% RSLogix 500 project SERVO VALVE CONTROL_BAK046.RSS, saved by version 8.30.00.16 %
PROJECT "UNTITLED"    % processor: Bul.1763 MicroLogix 1100 Series B %

PROGRAM FILES
  LAD 2 "MAIN"  4 rungs
  LAD 3 "DIGITAL IO"  8 rungs
  LAD 4 "CONTROLS"  8 rungs
  LAD 5 "POSITION"  6 rungs

DATA FILES
  O0 OUTPUT  4 elements
  I1 INPUT  6 elements
  S2 STATUS  66 elements
  B3 BINARY  12 elements
  T4 TIMER  3 elements
  C5 COUNTER  1 elements
  R6 CONTROL  1 elements
  N7 INTEGER  2 elements
  F8 FLOAT  1 elements

LADDER 2 "MAIN"
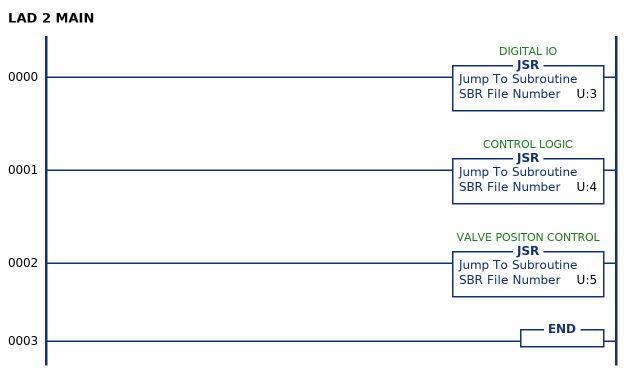
% Rung: 0 %
SOR JSR U:3 EOR
%   U:3  "DIGITAL IO" %
% Rung: 1 %
SOR JSR U:4 EOR
%   U:4  "CONTROL LOGIC" %
% Rung: 2 %
SOR JSR U:5 EOR
%   U:5  "VALVE POSITON CONTROL" %
% Rung: 3 %
SOR END EOR

LADDER 3 "DIGITAL IO"
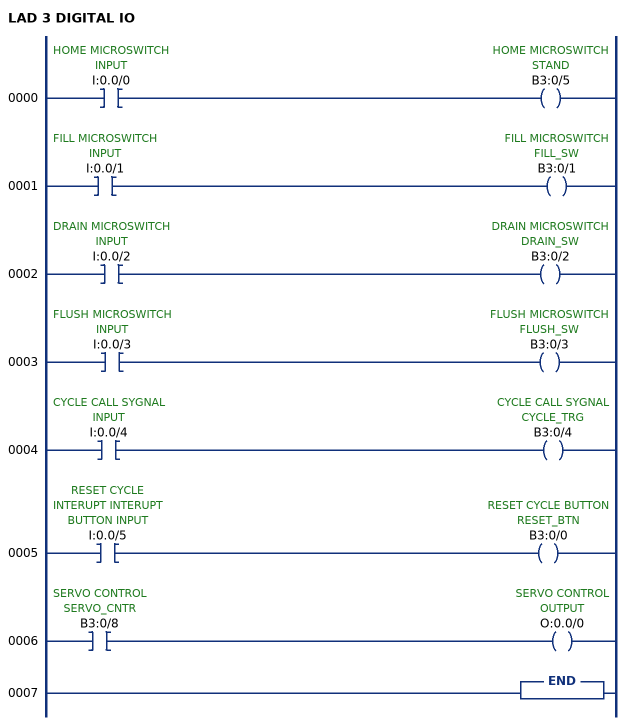
% Rung: 0 %
SOR XIC I:0.0/0 OTE B3:0/5 EOR
%   I:0.0/0  "HOME MICROSWITCH INPUT" %
%   B3:0/5  STAND  "HOME MICROSWITCH" %
% Rung: 1 %
SOR XIC I:0.0/1 OTE B3:0/1 EOR
%   I:0.0/1  "FILL MICROSWITCH INPUT" %
%   B3:0/1  FILL_SW  "FILL MICROSWITCH" %
% Rung: 2 %
SOR XIC I:0.0/2 OTE B3:0/2 EOR
%   I:0.0/2  "DRAIN MICROSWITCH INPUT" %
%   B3:0/2  DRAIN_SW  "DRAIN MICROSWITCH" %
% Rung: 3 %
SOR XIC I:0.0/3 OTE B3:0/3 EOR
%   I:0.0/3  "FLUSH MICROSWITCH INPUT" %
%   B3:0/3  FLUSH_SW  "FLUSH MICROSWITCH" %
% Rung: 4 %
SOR XIC I:0.0/4 OTE B3:0/4 EOR
%   I:0.0/4  "CYCLE CALL SYGNAL INPUT" %
%   B3:0/4  CYCLE_TRG  "CYCLE CALL SYGNAL" %
% Rung: 5 %
SOR XIC I:0.0/5 OTE B3:0/0 EOR
%   I:0.0/5  "RESET CYCLE INTERUPT INTERUPT BUTTON INPUT" %
%   B3:0/0  RESET_BTN  "RESET CYCLE BUTTON" %
% Rung: 6 %
SOR XIC B3:0/8 OTE O:0.0/0 EOR
%   B3:0/8  SERVO_CNTR  "SERVO CONTROL" %
%   O:0.0/0  "SERVO CONTROL OUTPUT" %
% Rung: 7 %
SOR END EOR

LADDER 4 "CONTROLS"
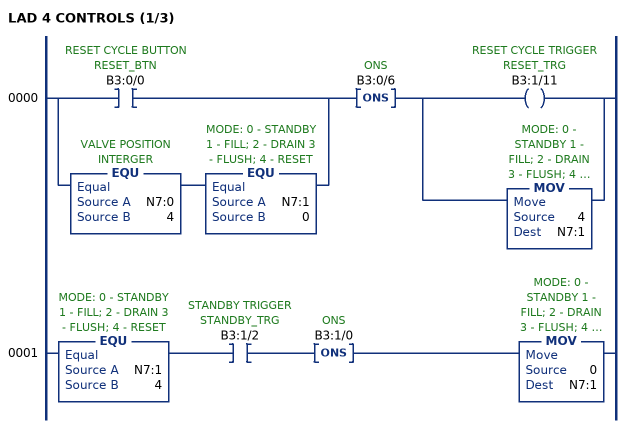
% Rung: 0 %
SOR BST XIC B3:0/0 NXB EQU N7:0 4 EQU N7:1 0 BND ONS B3:0/6 BST OTE B3:1/11 NXB MOV 4 N7:1 BND EOR
%   B3:0/0  RESET_BTN  "RESET CYCLE BUTTON" %
%   N7:0  "VALVE POSITION INTERGER" %
%   N7:1  "MODE: 0 - STANDBY 1 - FILL; 2 - DRAIN 3 - FLUSH; 4 - RESET" %
%   B3:0/6  "ONS" %
%   B3:1/11  RESET_TRG  "RESET CYCLE TRIGGER" %
% Rung: 1 %
SOR EQU N7:1 4 XIC B3:1/2 ONS B3:1/0 MOV 0 N7:1 EOR
%   N7:1  "MODE: 0 - STANDBY 1 - FILL; 2 - DRAIN 3 - FLUSH; 4 - RESET" %
%   B3:1/2  STANDBY_TRG  "STANDBY TRIGGER" %
%   B3:1/0  "ONS" %

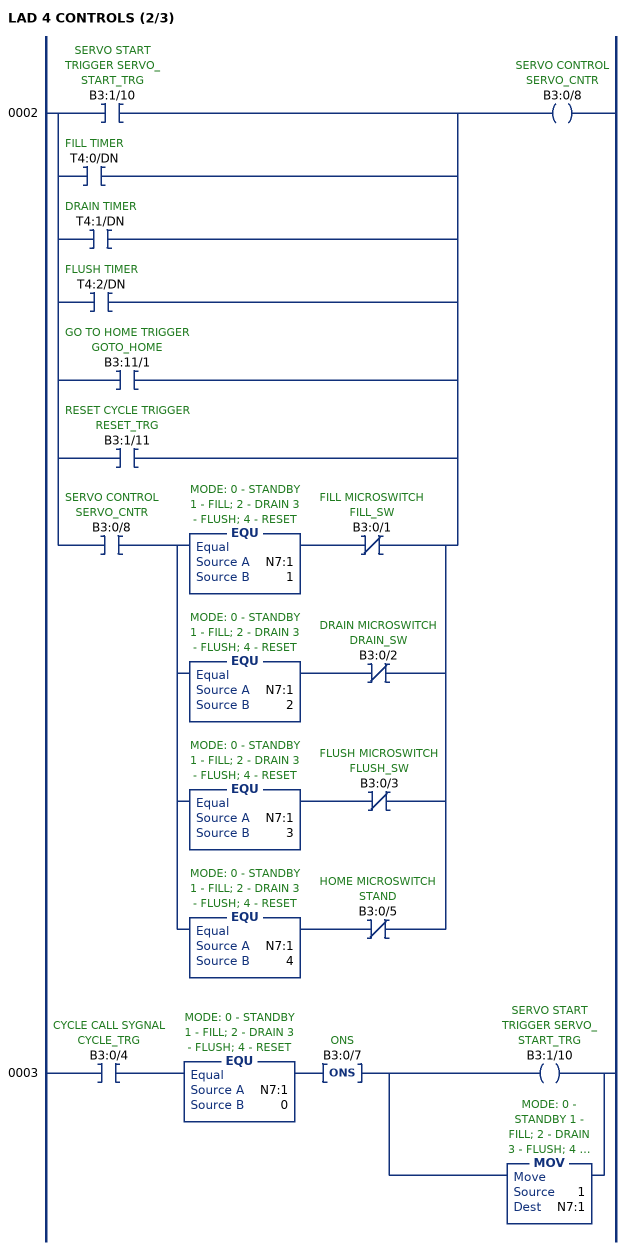
% Rung: 2 %
SOR BST BST XIC B3:1/10 NXB XIC T4:0/DN NXB XIC T4:1/DN NXB XIC T4:2/DN NXB XIC B3:11/1 NXB XIC B3:1/11 BND NXB XIC B3:0/8 BST EQU N7:1 1 XIO B3:0/1 NXB EQU N7:1 2 XIO B3:0/2 NXB EQU N7:1 3 XIO B3:0/3 NXB EQU N7:1 4 XIO B3:0/5 BND BND OTE B3:0/8 EOR
%   B3:1/10  SERVO_START_TRG  "SERVO START TRIGGER" %
%   T4:0  "FILL TIMER" %
%   T4:1  "DRAIN TIMER" %
%   T4:2  "FLUSH TIMER" %
%   B3:11/1  GOTO_HOME  "GO TO HOME TRIGGER" %
%   B3:1/11  RESET_TRG  "RESET CYCLE TRIGGER" %
%   B3:0/8  SERVO_CNTR  "SERVO CONTROL" %
%   N7:1  "MODE: 0 - STANDBY 1 - FILL; 2 - DRAIN 3 - FLUSH; 4 - RESET" %
%   B3:0/1  FILL_SW  "FILL MICROSWITCH" %
%   B3:0/2  DRAIN_SW  "DRAIN MICROSWITCH" %
%   B3:0/3  FLUSH_SW  "FLUSH MICROSWITCH" %
%   B3:0/5  STAND  "HOME MICROSWITCH" %
% Rung: 3 %
SOR XIC B3:0/4 EQU N7:1 0 ONS B3:0/7 BST OTE B3:1/10 NXB MOV 1 N7:1 BND EOR
%   B3:0/4  CYCLE_TRG  "CYCLE CALL SYGNAL" %
%   N7:1  "MODE: 0 - STANDBY 1 - FILL; 2 - DRAIN 3 - FLUSH; 4 - RESET" %
%   B3:0/7  "ONS" %
%   B3:1/10  SERVO_START_TRG  "SERVO START TRIGGER" %

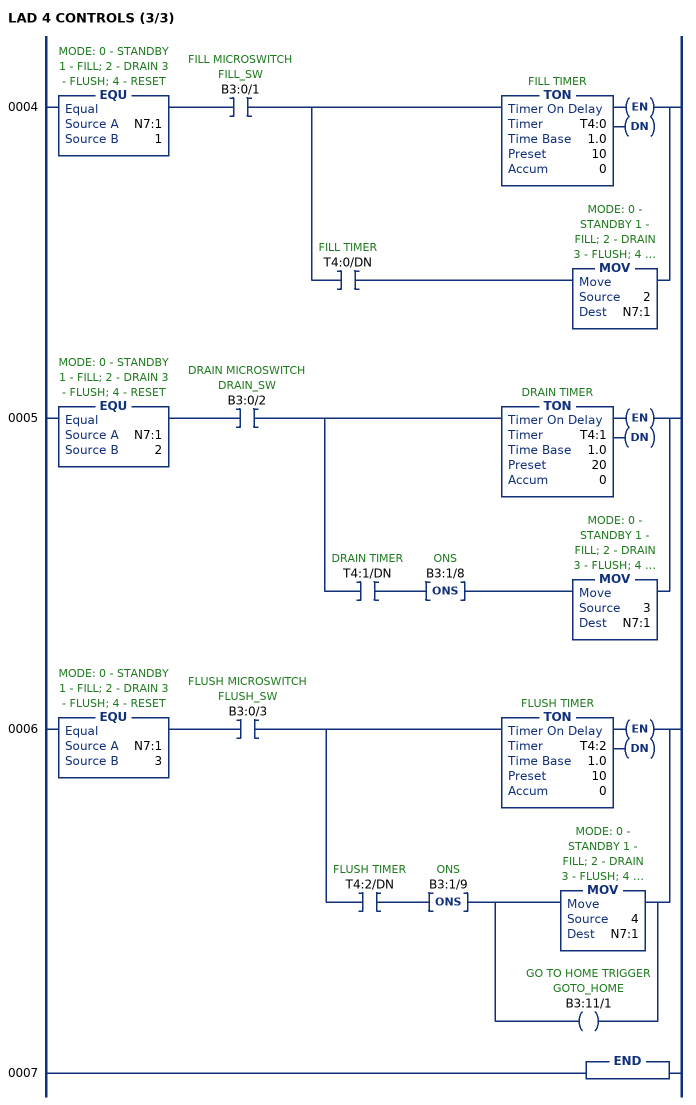
% Rung: 4 %
SOR EQU N7:1 1 XIC B3:0/1 BST TON T4:0 1.0 10 0 NXB XIC T4:0/DN MOV 2 N7:1 BND EOR
%   N7:1  "MODE: 0 - STANDBY 1 - FILL; 2 - DRAIN 3 - FLUSH; 4 - RESET" %
%   B3:0/1  FILL_SW  "FILL MICROSWITCH" %
%   T4:0  "FILL TIMER" %
% Rung: 5 %
SOR EQU N7:1 2 XIC B3:0/2 BST TON T4:1 1.0 20 0 NXB XIC T4:1/DN ONS B3:1/8 MOV 3 N7:1 BND EOR
%   N7:1  "MODE: 0 - STANDBY 1 - FILL; 2 - DRAIN 3 - FLUSH; 4 - RESET" %
%   B3:0/2  DRAIN_SW  "DRAIN MICROSWITCH" %
%   T4:1  "DRAIN TIMER" %
%   B3:1/8  "ONS" %
% Rung: 6 %
SOR EQU N7:1 3 XIC B3:0/3 BST TON T4:2 1.0 10 0 NXB XIC T4:2/DN ONS B3:1/9 BST MOV 4 N7:1 NXB OTE B3:11/1 BND BND EOR
%   N7:1  "MODE: 0 - STANDBY 1 - FILL; 2 - DRAIN 3 - FLUSH; 4 - RESET" %
%   B3:0/3  FLUSH_SW  "FLUSH MICROSWITCH" %
%   T4:2  "FLUSH TIMER" %
%   B3:1/9  "ONS" %
%   B3:11/1  GOTO_HOME  "GO TO HOME TRIGGER" %
% Rung: 7 %
SOR END EOR

LADDER 5 "POSITION"
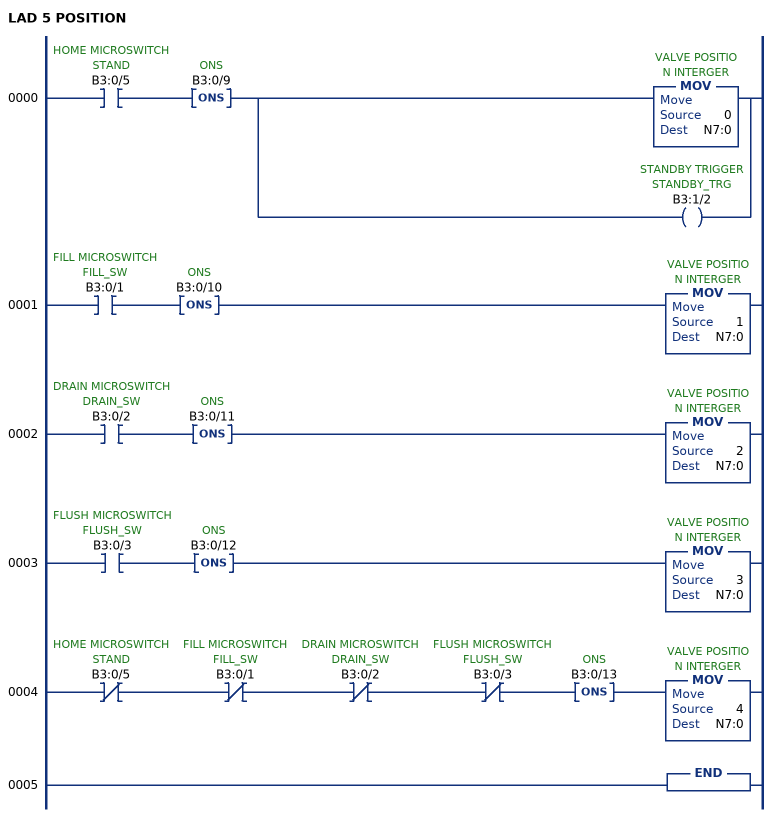
% Rung: 0 %
SOR XIC B3:0/5 ONS B3:0/9 BST MOV 0 N7:0 NXB OTE B3:1/2 BND EOR
%   B3:0/5  STAND  "HOME MICROSWITCH" %
%   B3:0/9  "ONS" %
%   N7:0  "VALVE POSITION INTERGER" %
%   B3:1/2  STANDBY_TRG  "STANDBY TRIGGER" %
% Rung: 1 %
SOR XIC B3:0/1 ONS B3:0/10 MOV 1 N7:0 EOR
%   B3:0/1  FILL_SW  "FILL MICROSWITCH" %
%   B3:0/10  "ONS" %
%   N7:0  "VALVE POSITION INTERGER" %
% Rung: 2 %
SOR XIC B3:0/2 ONS B3:0/11 MOV 2 N7:0 EOR
%   B3:0/2  DRAIN_SW  "DRAIN MICROSWITCH" %
%   B3:0/11  "ONS" %
%   N7:0  "VALVE POSITION INTERGER" %
% Rung: 3 %
SOR XIC B3:0/3 ONS B3:0/12 MOV 3 N7:0 EOR
%   B3:0/3  FLUSH_SW  "FLUSH MICROSWITCH" %
%   B3:0/12  "ONS" %
%   N7:0  "VALVE POSITION INTERGER" %
% Rung: 4 %
SOR XIO B3:0/5 XIO B3:0/1 XIO B3:0/2 XIO B3:0/3 ONS B3:0/13 MOV 4 N7:0 EOR
%   B3:0/5  STAND  "HOME MICROSWITCH" %
%   B3:0/1  FILL_SW  "FILL MICROSWITCH" %
%   B3:0/2  DRAIN_SW  "DRAIN MICROSWITCH" %
%   B3:0/3  FLUSH_SW  "FLUSH MICROSWITCH" %
%   B3:0/13  "ONS" %
%   N7:0  "VALVE POSITION INTERGER" %
% Rung: 5 %
SOR END EOR

OTHER DOCUMENTED ADDRESSES
  B3:0/14  "ONS"
  B3:0/15  "ONS"
  B3:1/1  "ONS"
  B3:1/3  FILL_TRG  "FILL TRIGGER"
  B3:1/4  GOTO_DRAIN  "GOTO DRAIN TRIGGER"
  B3:1/5  DRAIN_TRG  "DRAIN TRIGGER"
  B3:1/6  FLUSH_TRG  "FLUSH TRIGGER"
  B3:1/7  GOTO_FLUSH  "GOTO FLUSH TRIGGER"
  B4:1/4  "DRAIN TRIGGER"
  B4:1/5  "FLUSH TRIGGER"

DATA TABLE (non-zero values as saved)
DATA B3
% B3:0 % 0X0280 0X0000 0X0000 0X0000 0X0000 0X0000 0X0000 0X0000 0X0000 0X0000
DATA T4
% .PRE .ACC %
% T4:0 % 10 0
% T4:1 % 20 0
% T4:2 % 10 0
